TYPE ST_Sequence_Sts :
STRUCT
	not_started : BIT;
	started		: BIT;
	completed	: BIT;
	error		: BIT;
END_STRUCT
END_TYPE

(* stored: Version 1.1.0.1, ProductVersion 3.1.4024.12
   DUT ST_Sequence_Sts: Id {3cccb815-bf5c-4022-b7df-33ab18217ab0} *)
